(* IEC 61131-3 sources: Lasal/CPU_5344_V01/Class/AbsoluteIt, 1 file *)

(* ---- AbsoluteIt.st ---- *)
(*!
<Class
	Name               = "AbsoluteIt"
	Revision           = "0.0"
	RealtimeTask       = "false"
	CyclicTask         = "false"
	BackgroundTask     = "false"
	Sigmatek           = "false"
	OSInterface        = "false"
	HighPriority       = "false"
	Automatic          = "false"
	UpdateMode         = "Prescan"
	SharedCommandTable = "true"
	Objectsize         = "(284,120)">
	<Channels>
		<Server Name="ClassSvr" Visualized="false" Initialize="false" WriteProtected="false" Retentive="false"/>
		<Client Name="AnaOut" Required="true" Internal="false"/>
	</Channels>
</Class>
*)
AbsoluteIt : CLASS
  //Servers:
	ClassSvr 	: SvrChCmd_DINT;
  //Clients:
	AnaOut 	: CltCh_DINT;
  //Variables:
  //Functions:

	FUNCTION VIRTUAL GLOBAL ClassSvr::Write
		VAR_INPUT
			input (EAX) 	: DINT;
		END_VAR
		VAR_OUTPUT
			result (EAX) 	: DINT;
		END_VAR;
  //Tables:
	FUNCTION @STD
		VAR_OUTPUT
			ret_code	: CONFSTATES;
		END_VAR;
	FUNCTION GLOBAL TAB @CT_;
END_CLASS;

FUNCTION VIRTUAL GLOBAL AbsoluteIt::ClassSvr::Write
	VAR_INPUT
		input (EAX) 	: DINT;
	END_VAR
	VAR_OUTPUT
		result (EAX) 	: DINT;
	END_VAR

	ClassSvr := input;
  AnaOut := abs(ClassSvr);
  AnaOut.Write(input:=AnaOut);
	result := ClassSvr;

END_FUNCTION
